PROGRAM P_Example_2
VAR
	bStart, bPause 		: BOOL; 
	tSet_Time 			: TIME := T#1M; 
	tElapsed_RTime 		: TIME; 
	bElapsed_RTime 		: BOOL; 
	fbRTimer 			: FB_RTimer;
END_VAR

fbRTimer(bStart := bStart, bPause := bPause, tSet := tSet_Time,  
		 bElapsed => bElapsed_RTime, tElapsed => tElapsed_RTime);

END_PROGRAM

(* stored: Version 1.1.0.1, ProductVersion 3.1.4024.4
   POU P_Example_2: Id {c9fa6007-1c07-48f6-85a4-bf08c2520e2c}, SpecialFunc None *)
